KUKA KRL program: EXIT_BATT.src, EXIT_BATT.dat

--- EXIT_BATT.src ---
&ACCESS RVP2
&REL 13
&PARAM EDITMASK = *
&PARAM TEMPLATE = C:\KRC\Roboter\Template\vorgabe
DEF EXIT_BATT( )

END

GLOBAL DEF DoAbortLiquidTest ( )
  ; Subroutine to stop and cancel current
  ; LIN P40:{x 0,y 0,z -250,a 0,b 0,c 0}

  INTERRUPT OFF 96
  WAIT SEC 0.1
  $OUT[241]=FALSE
  $OUT[242]=TRUE
  WAIT SEC 0.5
  $OUT[242]=FALSE
   LIN_REL {Y -50,z -400}
  WAIT SEC 0.1
  INTERRUPT ON 96
END

--- EXIT_BATT.dat ---
&ACCESS RVP2
&REL 13
&PARAM EDITMASK = *
&PARAM TEMPLATE = C:\KRC\Roboter\Template\vorgabe
DEFDAT  EXIT_BATT PUBLIC
;FOLD EXTERNAL DECLARATIONS;%{PE}%MKUKATPBASIS,%CEXT,%VCOMMON,%P
;FOLD GRIPPERTECH EXT
EXT  H50 (INT  :IN,INT  :IN,INT  :IN,GRP_TYP  :IN )
;ENDFOLD (GRIPPERTECH EXT)
;FOLD SPOTTECH EXT
EXT  USERSPOT (S_COMMAND  :IN,SPOT_TYPE  :IN )
;ENDFOLD (SPOTTECH EXT)
;FOLD BASISTECH EXT;%{PE}%MKUKATPBASIS,%CEXT,%VEXT,%P
EXT  BAS (BAS_COMMAND  :IN,REAL  :IN )
DECL INT SUCCESS
;ENDFOLD (BASISTECH EXT)
;FOLD USER EXT;%{E}%MKUKATPUSER,%CEXT,%VEXT,%P
;Make your modifications here
GLOBAL BOOL DoAbort1=FALSE

ENDDAT
